FUNCTION_BLOCK FB_PneumaticAxis IMPLEMENTS I_MotionAxis
VAR_INPUT
END_VAR
VAR_OUTPUT
END_VAR
VAR
END_VAR

{warning 'Add method implementation '}
METHOD CalibrateEncValue
END_METHOD

{warning 'Add method implementation '}
METHOD EncSaveRestore
END_METHOD

{warning 'Add property implementation'}
PROPERTY Error : BOOL
GET
END_GET
END_PROPERTY

{warning 'Add property implementation'}
PROPERTY ErrorID : BOOL
GET
END_GET
END_PROPERTY

{warning 'Add method implementation '}
METHOD GearIn
END_METHOD

{warning 'Add method implementation '}
METHOD GearOut
END_METHOD

{warning 'Add method implementation '}
METHOD GetAxisRef : REFERENCE TO AXIS_REF
END_METHOD

{warning 'Add method implementation '}
METHOD GetPowerOverride : LREAL
END_METHOD

{warning 'Add method implementation '}
METHOD Halt
VAR_INPUT
    Deceleration	: LREAL := 0.0;
    Jerk	: LREAL := 0.0;
    BufferMode	: MC_BufferMode := .MC_BufferMode.MC_Aborting;
END_VAR
VAR_OUTPUT
    Done	: BOOL;
    Busy	: BOOL;
    Active	: BOOL;
    CommandAborted	: BOOL;
    Error	: BOOL;
    ErrorID	: UDINT;
    ErrorStr	: T_MaxString;
END_VAR
END_METHOD

{warning 'Add property implementation'}
PROPERTY HaltBusy : BOOL
GET
END_GET
END_PROPERTY

{warning 'Add property implementation'}
PROPERTY HaltDone : BOOL
GET
END_GET
END_PROPERTY

{warning 'Add property implementation'}
PROPERTY HaltError : BOOL
GET
END_GET
END_PROPERTY

{warning 'Add property implementation'}
PROPERTY HaltErrorID : UDINT
GET
END_GET
END_PROPERTY

{warning 'Add method implementation '}
METHOD Home
VAR_INPUT
    Position : LREAL := DEFAULT_HOME_POSITION;
    HomingMode : MC_HomingMode := MC_DefaultHoming;
END_VAR
VAR_OUTPUT
    Done	: BOOL;
    Busy	: BOOL;
    Active	: BOOL;
    CommandAborted	: BOOL;
    Error	: BOOL;
    ErrorID	: UDINT;
    ErrorStr	: T_MaxString;
END_VAR
END_METHOD

{warning 'Add property implementation'}
PROPERTY HomeBusy : BOOL
GET
END_GET
END_PROPERTY

{warning 'Add property implementation'}
PROPERTY HomeDone : BOOL
GET
END_GET
END_PROPERTY

{warning 'Add property implementation'}
PROPERTY MeasuredAcceleration : LREAL
GET
END_GET
END_PROPERTY

{warning 'Add property implementation'}
PROPERTY MeasuredPosition : LREAL
GET
END_GET
END_PROPERTY

{warning 'Add property implementation'}
PROPERTY MeasuredVelocity : LREAL
GET
END_GET
END_PROPERTY

{warning 'Add method implementation '}
METHOD MoveAbsolute
VAR_INPUT
    Position	: LREAL;
    Velocity	: LREAL;
    Acceleration	: LREAL := 0.0;
    Deceleration	: LREAL := 0.0;
    Jerk	: LREAL := 0.0;
    BufferMode	: MC_BufferMode := .MC_BufferMode.MC_Aborting;
END_VAR
VAR_OUTPUT
    Done	: BOOL;
    Busy	: BOOL;
    Active	: BOOL;
    CommandAborted	: BOOL;
    Error	: BOOL;
    ErrorID	: UDINT;
    ErrorStr	: T_MaxString;
END_VAR
END_METHOD

{warning 'Add property implementation'}
PROPERTY MoveAbsoluteBusy : BOOL
GET
END_GET
END_PROPERTY

{warning 'Add property implementation'}
PROPERTY MoveAbsoluteDone : BOOL
GET
END_GET
END_PROPERTY

{warning 'Add property implementation'}
PROPERTY MoveAbsoluteError : BOOL
GET
END_GET
END_PROPERTY

{warning 'Add property implementation'}
PROPERTY MoveAbsoluteErrorID : UDINT
GET
END_GET
END_PROPERTY

{warning 'Add property implementation'}
PROPERTY MoveAbsoluteTargetAcceleration : LREAL
GET
END_GET
END_PROPERTY

{warning 'Add property implementation'}
PROPERTY MoveAbsoluteTargetDeceleration : LREAL
GET
END_GET
END_PROPERTY

{warning 'Add property implementation'}
PROPERTY MoveAbsoluteTargetJerk : LREAL
GET
END_GET
END_PROPERTY

{warning 'Add property implementation'}
PROPERTY MoveAbsoluteTargetPosition : LREAL
GET
END_GET
END_PROPERTY

{warning 'Add property implementation'}
PROPERTY MoveAbsoluteTargetVelocity : LREAL
GET
END_GET
END_PROPERTY

{warning 'Add property implementation'}
PROPERTY MoveBusy : BOOL
GET
END_GET
END_PROPERTY

{warning 'Add property implementation'}
PROPERTY MoveDone : BOOL
GET
END_GET
END_PROPERTY

{warning 'Add property implementation'}
PROPERTY NegativeMotionIsEnabled : BOOL
GET
END_GET
END_PROPERTY

{warning 'Add property implementation'}
PROPERTY PositiveMotionIsEnabled : BOOL
GET
END_GET
END_PROPERTY

{warning 'Add method implementation '}
METHOD Power
VAR_INPUT
    Enable	: BOOL;
    Enable_Positive	: BOOL;
    Enable_Negative	: BOOL;
    (* in percent from 0 to 100 *)
    Override	: LREAL := 100.0;
    BufferMode	: MC_BufferMode := .MC_BufferMode.MC_Aborting;
END_VAR
VAR_OUTPUT
    Status	: BOOL;
    Busy	: BOOL;
    Active	: BOOL;
    Error	: BOOL;
    ErrorID	: UDINT;
    ErrorStr	: T_MaxString;
END_VAR
END_METHOD

{warning 'Add property implementation'}
PROPERTY PowerError : BOOL
GET
END_GET
END_PROPERTY

{warning 'Add property implementation'}
PROPERTY PowerErrorID : UDINT
GET
END_GET
END_PROPERTY

{warning 'Add property implementation'}
PROPERTY PowerIsEnabled : BOOL
GET
END_GET
END_PROPERTY

{warning 'Add property implementation'}
PROPERTY PowerOverride : LREAL
GET
END_GET
END_PROPERTY

{warning 'Add property implementation'}
PROPERTY PowerStatus : BOOL
GET
END_GET
END_PROPERTY

{warning 'Add method implementation '}
METHOD Reset
VAR_OUTPUT
    Done	: BOOL;
    Busy	: BOOL;
    Error	: BOOL;
    ErrorID	: UDINT;
    ErrorStr	: T_MaxString;
END_VAR
END_METHOD

{warning 'Add property implementation'}
PROPERTY SetpointAcceleration : LREAL
GET
END_GET
END_PROPERTY

{warning 'Add property implementation'}
PROPERTY SetpointJerk : LREAL
GET
END_GET
END_PROPERTY

{warning 'Add property implementation'}
PROPERTY SetpointPosition : LREAL
GET
END_GET
END_PROPERTY

{warning 'Add property implementation'}
PROPERTY SetpointVelocity : LREAL
GET
END_GET
END_PROPERTY

{warning 'Add method implementation '}
METHOD SetPowerOverride
VAR_INPUT
    (* in percent from 0 to 100 *)
    Override	: LREAL;
END_VAR
VAR_OUTPUT
    Status	: BOOL;
    Busy	: BOOL;
    Active	: BOOL;
    Error	: BOOL;
    ErrorID	: UDINT;
    ErrorStr	: T_MaxString;
END_VAR
END_METHOD

END_FUNCTION_BLOCK

(* stored: Version 1.1.0.1
   POU FB_PneumaticAxis: Id {e0eb4b14-2043-42ba-85e3-bf27d0e557c3}, SpecialFunc None
   Method CalibrateEncValue: Id {fe167c0d-f488-4318-b7c4-3b46544f8bb2}
   Method EncSaveRestore: Id {7797e056-c75d-4ac4-ad03-80c3806b726e}
   Property Error: Id {a78a81a3-1783-4065-a7db-61177e6b5f5c}
   Get Get: Id {0b8cb910-68e1-44a0-b3d0-02315b48a363}
   Property ErrorID: Id {abc3ebdb-4ff8-465c-a362-883e97bbb5df}
   Get Get: Id {54148e71-3368-4bd8-86d5-476ff522cb9c}
   Method GearIn: Id {ca2dc6b4-a648-4084-bbbf-76a814f1e5a2}
   Method GearOut: Id {6996a470-5098-4549-9a0b-e69a30f09d06}
   Method GetAxisRef: Id {e3665c87-1ba4-4099-88d3-d9b640f8d4ca}
   Method GetPowerOverride: Id {334bf9e4-ed2c-468f-bfd5-1f8dd5fca106}
   Method Halt: Id {af000cf0-4a65-4f07-a058-846e832b3d08}
   Property HaltBusy: Id {633b3062-1c92-45b0-8631-660f42363d1d}
   Get Get: Id {4b096186-1d2f-47c7-9fba-30383b44625d}
   Property HaltDone: Id {64abeddd-b975-431b-bdf2-8cc261a47326}
   Get Get: Id {4e6d97fd-63d3-402d-b474-80b22628207e}
   Property HaltError: Id {03e743a7-dd7b-45a0-99f3-cb4155792c6f}
   Get Get: Id {3c9073c3-dde6-4107-9535-d66889d9cfa8}
   Property HaltErrorID: Id {a5ca4f59-35af-4247-b4d3-f2b16326cd47}
   Get Get: Id {c2fedc2c-f493-49b5-b262-a63ad5280e03}
   Method Home: Id {74b22abb-7acd-4ef8-8d71-6953bcd77630}
   Property HomeBusy: Id {49cafa39-6135-40e9-bcc7-d416a05be7f3}
   Get Get: Id {a50107bf-6314-4145-a969-c387fc1df784}
   Property HomeDone: Id {a81ce99f-afa5-4363-9112-a0828aab461a}
   Get Get: Id {2daaeb4e-c087-4759-b2e5-720a4bfe9ebc}
   Property MeasuredAcceleration: Id {689e2442-f916-4f22-a8a8-b6995730bd63}
   Get Get: Id {094fb608-780e-4e12-adaf-1ce79c520d9a}
   Property MeasuredPosition: Id {801eefa4-fa82-40b5-9d5d-7a36378d7441}
   Get Get: Id {fdf2cc46-a5e0-4485-ba1f-5bbec43c1544}
   Property MeasuredVelocity: Id {cb8ba19f-1ed5-43d2-8630-c4fa77aa0574}
   Get Get: Id {86c3a9cc-494f-4387-9d3b-8bd1538c8664}
   Method MoveAbsolute: Id {0669991e-7faf-4ac7-9883-fcc16749394c}
   Property MoveAbsoluteBusy: Id {74c9aef3-7a90-4529-98da-fc24f8e69512}
   Get Get: Id {0b6efa0e-1b74-4dfb-9ff2-d8986cc437db}
   Property MoveAbsoluteDone: Id {474be2c2-841e-430c-95d6-0f2ed1862686}
   Get Get: Id {f750ab09-dd5c-410a-81b9-9b2e3c36f685}
   Property MoveAbsoluteError: Id {89a8bf2b-4924-43cb-97d2-80b8f78b0f34}
   Get Get: Id {35075af7-1c88-404d-aee5-24c34181df94}
   Property MoveAbsoluteErrorID: Id {2d8fcad7-2e8b-439e-9925-a3fed96f594c}
   Get Get: Id {d5f35bdc-ad1c-4005-9feb-8d1dc8b8d2b8}
   Property MoveAbsoluteTargetAcceleration: Id {c0f98dd1-096a-4bae-b143-be44fa211cc6}
   Get Get: Id {9585323e-4492-44c1-b383-0c2ee28d3ff6}
   Property MoveAbsoluteTargetDeceleration: Id {af9b5644-db93-4212-aa85-f50dfccc44b7}
   Get Get: Id {a67e3a22-b5f2-4cfb-91aa-f20e87b4bc20}
   Property MoveAbsoluteTargetJerk: Id {828148e6-d2b1-4cb8-a00a-76f123f5ebec}
   Get Get: Id {9ffaf1e4-9ebf-48df-bef6-d287d23f682b}
   Property MoveAbsoluteTargetPosition: Id {73b578bd-bdca-4e93-a567-63132a8528cd}
   Get Get: Id {79e606c2-dc71-43e1-80fc-e7088e3bd370}
   Property MoveAbsoluteTargetVelocity: Id {7f0f11b5-da84-4ebc-92b4-339931457070}
   Get Get: Id {3b7c95f5-0de7-414a-9857-4a1ebd0659ec}
   Property MoveBusy: Id {e3faad96-2fe5-4e3f-8bfc-f8521326939e}
   Get Get: Id {35b3c99b-a904-44e5-a25e-8debb6f4fdb6}
   Property MoveDone: Id {e0b80a72-8ebb-4150-843e-2865ee91b489}
   Get Get: Id {e55e50e3-a2a4-43a1-b7f0-81eac8731b2b}
   Property NegativeMotionIsEnabled: Id {f5f82dd5-89d6-431e-b05f-01d74dcc4bbf}
   Get Get: Id {67a24088-5c0b-44c3-86cd-e6e383412f7a}
   Property PositiveMotionIsEnabled: Id {537d6230-1e8d-4650-846e-0d63b9a574d9}
   Get Get: Id {e1dd3135-bcf9-4efc-bcb0-55c8db3a82b0}
   Method Power: Id {b2d25f6b-088e-4ac8-a1da-78cfc0505e5b}
   Property PowerError: Id {a510d09e-8b73-4272-b4a8-978ce7fd6072}
   Get Get: Id {38a0d2b0-aa09-4e07-bb5d-7f2b3a10d853}
   Property PowerErrorID: Id {eb9222a2-5119-4b4e-8fc5-f8a009dcf353}
   Get Get: Id {272c0c47-46f7-40d4-93ab-4c4569996628}
   Property PowerIsEnabled: Id {727c46f3-a2f4-4363-af3b-be57a79ba3e3}
   Get Get: Id {0e3b5b62-c66d-40f3-9253-fa491908912d}
   Property PowerOverride: Id {079526df-2c9f-497b-aa35-c674df0daab9}
   Get Get: Id {f342dd00-accd-4054-aa77-050a31c8bbed}
   Property PowerStatus: Id {373d50d7-76f5-4163-a97f-75b8d5ce2e58}
   Get Get: Id {571aca7a-b813-4021-a280-55c4cc60719e}
   Method Reset: Id {294f2062-ab27-4183-949a-b618b9d84b15}
   Property SetpointAcceleration: Id {a17023a0-983e-422b-9231-13d8380e6084}
   Get Get: Id {7fc448cb-fe5a-48ec-9c91-4441f41240e7}
   Property SetpointJerk: Id {ad472e92-0442-48f9-bbaa-be188c03e0f9}
   Get Get: Id {788ce13b-f080-4a33-bb36-b5c0dc5760bd}
   Property SetpointPosition: Id {408751d9-0f82-443e-b22d-c70e67f39e83}
   Get Get: Id {8a8a2170-f144-4724-90e4-ce2b9f126a98}
   Property SetpointVelocity: Id {bdd0a9bf-d5bc-456f-99ee-d6d2c510e030}
   Get Get: Id {bc19e35a-0b5b-4c13-bc09-070351a89e5b}
   Method SetPowerOverride: Id {227bd8a9-cc14-4744-bea4-3f77553c78be} *)
